TYPE ST_LaudaReadCommands_Cooling :
STRUCT
	CoolingMode	: STRING := 'IN_SP_02';
END_STRUCT
END_TYPE

(* stored: Version 1.1.0.1, ProductVersion 3.1.4024.13
   DUT ST_LaudaReadCommands_Cooling: Id {495a0683-f96e-41d2-8bc4-893801625e7d} *)
